(* CODESYS project LD_FB.xml

Project tree, tasks and I/O mapping:
  function block LD_FB [LD]
*)

// LD_FB
FUNCTION_BLOCK LD_FB
VAR_INPUT
	xStart : BOOL;
	xStop_NC : BOOL;
END_VAR
VAR_OUTPUT
	xPump : BOOL;
	xLamp : BOOL;
END_VAR
VAR
	
	
	
	timer : TON;
END_VAR

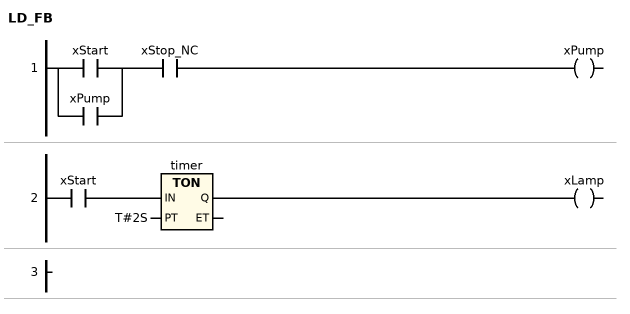
// NETWORK 1
xPump := (xStart OR xPump) AND xStop_NC;

// NETWORK 2
timer(IN := xStart, PT := T#2S); // TON
xLamp := timer.Q;

// NETWORK 3

END_FUNCTION_BLOCK
